FUNCTION_BLOCK FB_Sign_Test EXTENDS TcUnit.FB_TestSuite

TestCase('Sign Negative_1', fValue := -0.00001, fExpected:= -1);
TestCase('Sign Negative_2', fValue := -0.1, fExpected:= -1);
TestCase('Sign Negative_3', fValue := -1, fExpected:= -1);

TestCase('Sign Positive_1', fValue := 0, fExpected:= 1);
TestCase('Sign Positive_2', fValue := 0.00001, fExpected:= 1);
TestCase('Sign Positive_3', fValue := 0.1, fExpected:= 1);
TestCase('Sign Positive_4', fValue := 1, fExpected:= 1);

METHOD TestCase
VAR_INPUT
	sName : T_MaxString;	
	fValue : REAL; 
	fExpected : REAL;
END_VAR

VAR	
	fResult : REAL;
END_VAR
TEST(sName);
	
fResult := F_Sign(fValue);
AssertEquals(Expected := fExpected,
             Actual := fResult,
             Message := 'Result value is not correct');	
	 
TEST_FINISHED();
END_METHOD

END_FUNCTION_BLOCK

(* stored: Version 1.1.0.1, ProductVersion 3.1.4024.12
   POU FB_Sign_Test: Id {7fdae462-211d-06e1-0793-54b6355243c5}, SpecialFunc None
   Method TestCase: Id {dbae30a7-c218-0547-0ca3-ce305f478e4d} *)
